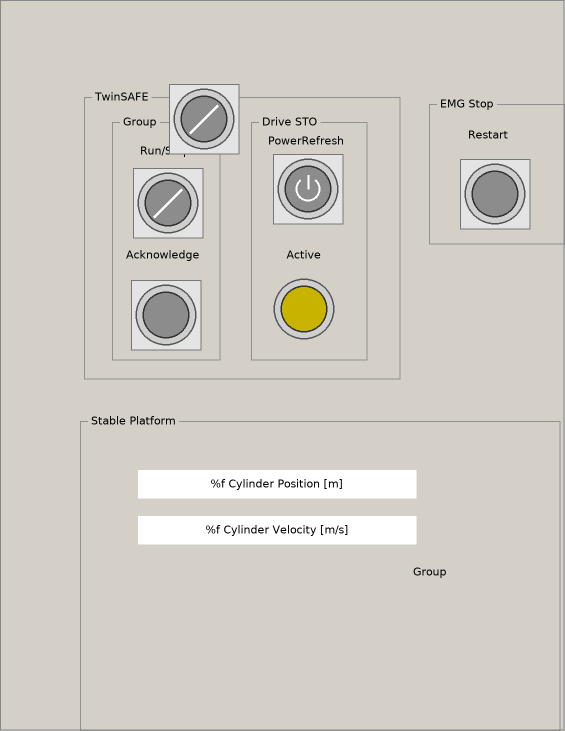
VISUALIZATION HMI  // 565x731
    GroupBox (84,89 316x290), "TwinSAFE"
        Label (268,468 156x30), "Group"
        Label (3,47 156x30), "Run/Stop"
        Label (1,151 156x30), "Acknowledge"
        GroupBox (28,25 108x246), "Group"
            RotarySwitch (21,54 70x70), variable: G_Safety_AXIS4.TwinSafeGroupRunStop, behaviour: TOGGLE, style: Switch-RotarySwitch-Gray
            PushSwitch (19,166 70x70), variable: G_Safety_AXIS4.TwinSafeGroupComErrAck, behaviour: TAP, style: Switch-PushSwitch-Gray
        Lamp1 (170,918 70x70), variable: G_Safety_AXIS4.ChA_STO_Active, style: Lamp-Lamp1-Yellow
        GroupBox (167,25 116x246), "Drive STO"
            RotarySwitch (-82,-30 70x70), behaviour: TOGGLE, style: Switch-RotarySwitch-Gray
            Lamp1 (18,160 70x70), variable: G_Safety_AXIS4.ChA_STO_Active, style: Lamp-Lamp1-Yellow
            PowerSwitch (22,40 70x70), variable: G_Safety_AXIS4.bWinchMotor24vDisable, behaviour: TAP, style: Switch-PowerSwitch-Gray
        Label (145,151 150x30), "Active"
        Label (147,37 150x30), "PowerRefresh"
    GroupBox (80,413 480x318), "Stable Platform"
        Textfield (57,56 280x30), "%f Cylinder Position [m]", text variable: G_StablePlatformScaledIO.fPistonPosition
        Textfield (57,102 280x30), "%f Cylinder Velocity [m/s]", text variable: G_StablePlatformScaledIO.fPistonVelocity
    GroupBox (429,96 136x148), "EMG Stop"
        PushSwitch (31,63 70x70), variable: G_Safety_AXIS4.EMGRestart, behaviour: TAP, style: Switch-PushSwitch-Gray
    Label (413,120 150x30), "Restart"
END_VISUALIZATION

(* stored: Version 1.1.0.1, ProductVersion 3.1.4024.12
   Visu HMI: Id {4fc9a593-5585-4c7b-9c87-b23c76f2039c} *)
